FUNCTION_BLOCK AUTOtimer
VAR_INPUT
	vrednost: BOOL;
	inpCas: TIME;
END_VAR
VAR_OUTPUT
	outCas: BOOL;
END_VAR
VAR
	TimerAutomatic: TOF;
END_VAR

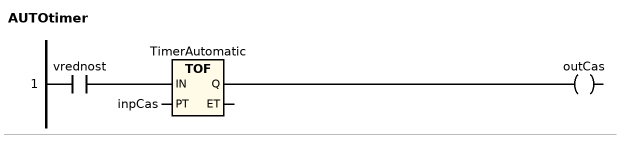
// NETWORK 1
TimerAutomatic(IN := vrednost, PT := inpCas); // TOF
outCas := TimerAutomatic.Q;

END_FUNCTION_BLOCK

(* stored: Version 1.1.0.1, ProductVersion 3.1.4024.15
   POU AUTOtimer: Id {043a6426-9f5f-4542-abc2-6383ac20737a}, SpecialFunc None *)
